(* PLC project Unnamed, Unknown Unnamed 1 *)
(* stored: creationDateTime 2024-05-08T15:05:08, modificationDateTime 2024-05-08T15:33:18 *)

PROGRAM Coil_and_Contact
  VAR
    Toggle_Switch : BOOL;
    Coil_1 : BOOL;
    Coil_2 : BOOL;
    Coil_3 : BOOL;
    Coil_4 : BOOL;
  END_VAR

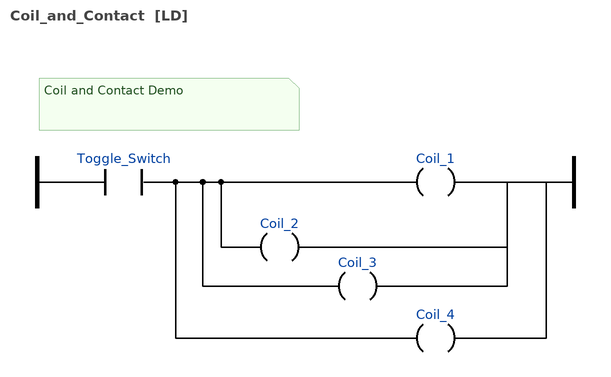
(* LD diagram, written out as Structured Text *)
(* Coil and Contact Demo *)
Coil_1 := Toggle_Switch;
Coil_2 := Toggle_Switch;
Coil_3 := Toggle_Switch;
Coil_4 := Toggle_Switch;
END_PROGRAM

CONFIGURATION Config0
  RESOURCE Res0 ON PLC
    TASK task0(INTERVAL := T#20ms, PRIORITY := 0);
    PROGRAM instance0 WITH task0 : Coil_and_Contact;
  END_RESOURCE
END_CONFIGURATION
